TYPE ST_HardSettings_PeakshaveBox:
STRUCT

END_STRUCT
END_TYPE

(* stored: Version 1.1.0.1, ProductVersion 3.1.4026.18
   DUT ST_HardSettings_PeakshaveBox: Id {2be4e1df-11fc-41a8-9be1-ac1d2c7fae57} *)
